// TIA Portal V18 export
TYPE "UDT_AHUSummaryAlarms"
// stored: IsFailsafeCompliant false
   STRUCT
      FrostAlarm : Array[1..3] of Bool;   // 0Active/Uack 0 - no blocking alarms/ 1- blocking alarms/ 2- frost alrm
      BlockingAlarm : Array[1..3] of Bool;
      HeaterPump : Array[1..3] of Bool;
      SAFAlarm : Array[1..3] of Bool;
      SAFilterAlarm : Array[1..3] of Bool;
   END_STRUCT;
END_TYPE
